// TIA Portal project "Temporizadores" (V16)

(* hardware
DEVICE "S7-1200 station_1"  S7-1200 Station
   slot 0: "Rack_0"  S7-1200 Rack  Rack  V1.0
   slot 1: "PLC_1"  CPU 1214C AC/DC/Rly  6ES7 214-1BG40-0XB0  V4.2
   slot 3: "DQ 4x24VDC_1"  DQ4 signal board (200 kHz)  6ES7 222-1BD30-0XB0  V1.0
*)

// ===== PLC "PLC_1"  CPU 1214C AC/DC/Rly =====

VAR_GLOBAL   // PLC tag table "Tabla de variables estándar"
   "TIMER" AT %MD0 : Time;
   "Tag_1" AT %I0.1 : Bool;
   "Tag_2" AT %I0.2 : Bool;
   "Tag_3" AT %Q0.7 : Bool;
   "Tag_4" AT %Q0.6 : Bool;
END_VAR

VAR_GLOBAL   // PLC tag table "Salidas"
   "Carga1" AT %Q0.1 : Bool;
   "Carga2" AT %Q0.2 : Bool;
   "Carga3" AT %Q0.3 : Bool;
END_VAR

VAR_GLOBAL   // PLC tag table "Entradas"
   "Arrancar" AT %I0.0 : Bool;
END_VAR

// folder: System blocks/Program resources

DATA_BLOCK "TM1"   // DB1
{ S7_Optimized_Access := 'TRUE' }
AUTHOR : Simatic
FAMILY : IEC
NAME : IEC_TMR
VERSION : 1.0
// stored: InstanceOfName IEC_TIMER
"IEC_TIMER"
BEGIN
END_DATA_BLOCK

DATA_BLOCK "TM2"   // DB2
{ S7_Optimized_Access := 'TRUE' }
AUTHOR : Simatic
FAMILY : IEC
NAME : IEC_TMR
VERSION : 1.0
// stored: InstanceOfName IEC_TIMER
"IEC_TIMER"
BEGIN
END_DATA_BLOCK

DATA_BLOCK "TM1.1"   // DB3
{ S7_Optimized_Access := 'TRUE' }
AUTHOR : Simatic
FAMILY : IEC
NAME : IEC_TMR
VERSION : 1.0
// stored: InstanceOfName IEC_TIMER
"IEC_TIMER"
BEGIN
END_DATA_BLOCK

// folder: (top level)

ORGANIZATION_BLOCK "Main"   // OB1, LAD, ProgramCycle
TITLE = "Main Program Sweep (Cycle)"
{ S7_Optimized_Access := 'TRUE' }
VERSION : 0.1
   VAR_INPUT
      Initial_Call : Bool;   // Initial call of this OB
      Remanence : Bool;   // =True, if remanent data are available
   END_VAR
BEGIN

REGION Network 1
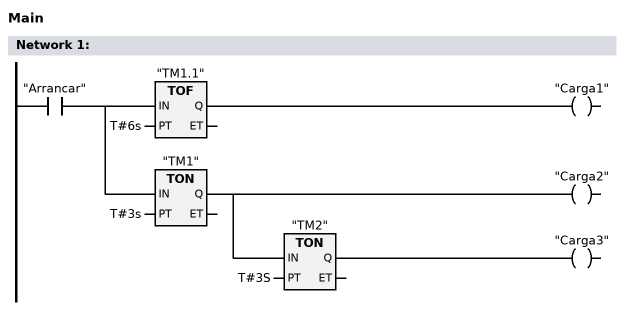
   "TM1.1".TOF(IN := "Arrancar", PT := T#6s);
   "Carga1" := "TM1.1".Q;
   "TM1".TON(IN := "Arrancar", PT := T#3s);
   "Carga2" := "TM1".Q;
   "TM2".TON(IN := "TM1".Q, PT := T#3S);
   "Carga3" := "TM2".Q;
END_REGION
END_ORGANIZATION_BLOCK